(* IEC 61131-3 sources: Industry-PLC-LLM/data/PLCBEAD_repo/PLCBEAD_PLCEmbed-main/PLC-BEAD/Source/GEB/HOUR_TO_TOD, 1 file *)

(* ---- HOUR_TO_TOD.ST ---- *)
FUNCTION _REAL_TO_UDINT:UDINT
	VAR_INPUT
		X :	REAL;
	END_VAR

	IF REAL_TO_UDINT(0.5) = UDINT#1 THEN
		_REAL_TO_UDINT := REAL_TO_UDINT(X);
	ELSIF X > 0.0 THEN
		_REAL_TO_UDINT := REAL_TO_UDINT(X+0.5);
	ELSIF X < 0.0 THEN
		_REAL_TO_UDINT := REAL_TO_UDINT(X-0.5);
	ELSE
		_REAL_TO_UDINT := UDINT#0;
	END_IF;

END_FUNCTION

FUNCTION HOUR_TO_TOD:UDINT

	VAR_INPUT
		IN :	REAL;
	END_VAR

	HOUR_TO_TOD := _REAL_TO_UDINT(IN * 3600000.00);

END_FUNCTION

PROGRAM program0
	VAR
		IN :	REAL;
		CEIL5_OUT : UDINT;
	END_VAR

  	CEIL5_OUT := HOUR_TO_TOD(IN);
END_PROGRAM
